{attribute 'pack_mode' := '1'}
TYPE TManDrivePos :
	STRUCT
		Teach			: BOOL	 := FALSE;
		TeachedPos		: LREAL;
		MoveToTeach	: TManButton;
	END_STRUCT
END_TYPE

(* stored: Version 1.1.0.1, ProductVersion 3.1.4022.12
   DUT TManDrivePos: Id {a87bb00a-93d3-4191-adaa-35d50fc11017} *)
